{attribute 'Tc2GvlVarNames'}
{attribute 'strict'}
//Stato Deposizione Layer
TYPE e_Stato_Layer :
(
	NOT_DEFINED					:= -1,
	LAYER_DA_DEPOSITARE			:= 0, 	(* Identifica che il deposito della Falda DEVE essere eseguito *)
	LAYER_DEPOSITATO			:= 1 	(* Identifica che il deposito della Falda E' AVVENUTO o NON DEVE essere eseguito *)
);
END_TYPE
//  NOT_DEFINED = '-1'

(* stored: Version 1.1.0.1, ProductVersion 3.1.4024.11
   EnumerationTextList e_Stato_Layer: Id {5c0c4fc2-5be5-42ad-a03d-c2e939012aa9} *)
